(* CODESYS project TU München_Base.project

Project tree, tasks and I/O mapping:
  Device : CODESYS Control Win V3, 3S - Smart Software Solutions GmbH, order no. 305021, version 3.5.10.0
    application project
      libraries: Tc2_Standard, 3.3.1.0 (Beckhoff Automation GmbH); Tc2_System, 3.4.14.0 (Beckhoff Automation GmbH); Tc3_Interfaces, 3.4.2.0 (Beckhoff Automation GmbH); Tc3_Module, 3.3.11.0 (Beckhoff Automation GmbH)
      task PlcTask (cyclic, interval t#200ms, priority 22) calls MAIN
      GVLs/
        global variables GVL
      POUs/
        OMAC/
          Data Structures/
            Enum/
              data type TDataType
              data type TDiagnosisState
              data type TOperation
              data type TOperationState
              data type TPositionTable
            Condition/
              function block Condition [ST]: value, name
          OMAC_PackML_State_Machine/
            Enums/
              data type State
            Function Blocks/
              function block UnitMode [ST]: Reset, Stop, Hold, Enter, Suspend, AllowsEntering, ActingStateCompleted, UnSuspend, Clear, Start, UnHold, NextState, Abort, AllowsLeaving, Name, SupportedStates, CurrentState, Active
              function block UnitModeManager [ST]: Register, FindMode, SwitchUnitMode, AllowsSwitchingTo, ActiveUnitModeNumber, ActiveUnitMode
              function block Test [ST]
            Interfaces/
              interface IUnitMode: Stop, Hold, Unhold, Abort, NextState, Suspend, Start, ActingStateCompleted, AllowsEntering, UnSuspend, Enter, Reset, Clear, Name, CurrentState, Active, AllowsLeaving, SupportedStates
              interface IPlant
          Interface/
            interface IModule: resetting, completing, starting, holding, aborting, unHolding, stopping, clearing, execute
        program MAIN [ST]
        CM/
          function block Conveyor1 [ST]: transportWPToRamp1, holding, clearing, aborting, resetting, completing, stopping, starting, execute, transportWPToStart, unHolding
          function block Crane [ST]: turnLeftToStack, unHolding, lift, clearing, completing, execute, starting, turnRightToStack, turnRightToStamp, intake, turnLeftToConveyor, turnRightToConveyor, lower, turnLeftToStamp, holding, stopping, aborting, resetting, release
          function block Stack [ST]: offer, resetting, release, aborting, clearing, holding, completing, wait, starting, unHolding, stopping, execute
          function block Stamp [ST]: wait, clearing, lower, offer, lift, aborting, starting, resetting, execute, completing, unHolding, holding, stopping, release
        ConditionObserver/
          function block ConditionObserver [ST]: addPositivePrecondition, addNegativePreAndPostcondition, addPositivePostcondition, addCondition, checkConditions, addObjectsFromBuffer
        DiagnosisModul/
          function block DiagnosisModule [ST]: executeFailureDiagnois
        EM/
          function block SortingPlant [ST]: execute, unHolding, aborting, stopping, completing, clearing, starting, resetting, holding
          function block StampingPlant [ST]: holding, aborting, resetting, unHolding, clearing, completing, stopping, starting, execute
        UN/
          function block PickAndPlaceUnit [ST]: resetting, execute, completing, starting, holding, aborting, unHolding, clearing, stopping
*)

// Device/project/POUs/OMAC/Data Structures/Enum/TDataType
{attribute 'strict' := ''}
TYPE TDataType :
(
	tGRAPH := 0,
	tOPERATION := 1
);
END_TYPE

// Device/project/POUs/OMAC/Data Structures/Enum/TDiagnosisState
TYPE TDiagnosisState :
(
	tNODIAGNOSISSTATE := 0,
	tDIAGNOSISSTEP1,
	tDIAGNOSISSTEP2,
	tDIAGNOSISSTEP3,
	tDIAGNOSISSTEP4,
	tDIAGNOSISSTEP5,
	tDIAGNOSISFINISHED
);
END_TYPE

// Device/project/POUs/OMAC/Data Structures/Enum/TOperation
TYPE TOperation :
(
	tOPERATING := 0,
	tFINISHED := 1,
	tERROR := 2,
	tNORESPONSE := 3
);
END_TYPE

// Device/project/POUs/OMAC/Data Structures/Enum/TOperationState
TYPE TOperationState :
(
	tNOSTATE := 0,
	tSTACKEXTENDCYLINDER,
	tSTACKRETRACTCYLINDER,
	tSTACKWAITFOREXTEND,
	tCRANELOWERATSTACK,
	tCRANEINTAKE,
	tCRANELIFTATSTACK,
	tCRANETURNTOSTAMP,
	tCRANELOWERATSTAMP,
	tCRANERELEASE,
	tCRANELIFTATSTAMP,
	tCRANETURNTOCONVEYOR,
	tCRANELOWERATCONVEYOR,
	tCRANELIFTATCONVEYOR,
	tSTAMPRELEASE,
	tSTAMPLOWER,
	tSTAMPWAIT,
	tSTAMPLIFT,
	tSTAMPOFFER,
	tSTAMPINGPLANTTRANSPORTWPTOSTAMP,
	tSTAMPINGPLANTPROVIDEWP,
	tSTAMPINGPLANTSTAMPWP,
	tSTAMPINGPLANTTRANSPORTWPTOCONVEYOR,
	tCONVEYOR1TRANSPORTWPTORAMP1,
	tSORTINGPLANTTRANSPORTWPTORAMP,
	tPPUSTAMPWP,
	tPPUSORTWP,
	tOPERATIONFINISHED
);
END_TYPE

// Device/project/POUs/OMAC/Data Structures/Enum/TPositionTable
TYPE TPositionTable :
(
	NOPOSITION := 0,
	POSITION1,
	POSITION2,
	POSITION3,
	POSITION4,
	POSITION5,
	POSITION6,
	POSITION7,
	POSITION8
);
END_TYPE

// Device/project/POUs/OMAC/OMAC_PackML_State_Machine/Enums/State
/// Machine states
TYPE State :
(
	/// Bit 0
	Stopped := 16#1,
	/// Bit 1
	Resetting := 16#2,
	/// Bit 2
	Idle := 16#4,
	/// Bit 3
	Starting := 16#8,
	/// Bit 4
	Execute := 16#10,
	/// Bit 5
	Holding := 16#20,
	/// Bit 6
	Held := 16#40,
	/// Bit 7
	UnHolding := 16#80,
	/// Bit 8
	Suspending := 16#100,
	/// Bit 9
	Suspended := 16#200,
	/// Bit 10
	UnSuspending := 16#400,
	/// Bit 11
	Completing := 16#800,
	/// Bit 12
	Complete := 16#1000,
	/// Bit 13
	Stopping := 16#2000,
	/// Bit 14
	Aborting := 16#4000,
	/// Bit 15
	Aborted := 16#8000,
	/// Bit 16
	Clearing := 16#10000,
	No := 0,
	All := 16#1FFFF,
	Invalid := 16#80000000
) DWORD;
END_TYPE

// Device/project/GVLs/GVL
VAR_GLOBAL
	in_MagazinStartknopf : BOOL;
	in_MagazinNotaus : BOOL;
	in_MagazinSchieberAusgefahren : BOOL;
	in_MagazinSchieberNichtAusgefahren : BOOL;
	in_MagazinInduktiverSensor : BOOL;
	in_MagazinOptischerSensor : BOOL;
	in_MagazinWerkstueckGriffbereit : BOOL;
	
	in_KranAngesaugt : BOOL;
	in_KranUnten : BOOL;
	in_KranOben : BOOL;
	in_KranZeigtAufStempel : BOOL;
	in_KranZeigtAufLaufband : BOOL;
	in_KranZeigtAufMagazin : BOOL;
	
	in_StempelSchieberAusgefahren  : BOOL;
	in_StempelSchieberEingefahren  : BOOL;
	in_StempelWerkstueckVorhanden  : BOOL;
	in_StempelOben  : BOOL;
	in_StempelUnten  : BOOL;
	
	in_Sortierband_LichttasterKranInterface  : BOOL;
	in_Sortierband_KapazitiverSensorKranInterface  : BOOL;
	in_Sortierband_InduktiverSensorPusher1  : BOOL;
	in_Sortierband_LichttasterPusher1  : BOOL;
	in_Sortierband_InduktiverSensorPusher2  : BOOL;
	in_Sortierband_LichttasterPusher2  : BOOL;
	in_Sortierband_LichttasterSlide3  : BOOL;
	in_Sortierband_Pusher1Ausgefahren  : BOOL;
	in_Sortierband_Pusher1Eingefahren  : BOOL;
	in_Sortierband_Pusher2Ausgefahren  : BOOL;
	in_Sortierband_Pusher2Eingefahren  : BOOL;
	in_Sortierband_Lichtschranke3  : BOOL;
	
	in_Magazin_SchalterManAuto  : BOOL;
	
	out_MagazinSchieber : BOOL;
	
	out_KranSenken : BOOL;
	out_KranVakuumAn : BOOL;
	out_KranDreheRechts : BOOL;
	out_KranDreheLinks : BOOL;
	
	out_StempelSchieberAusfahren  : BOOL;
	out_StempelSchieberEinfahren  : BOOL;
	out_StempelStempeln  : BOOL;
	out_StempelStempelnDruck  : INT;
	
	out_SortierbandDreheVorwaerts  : BOOL;
	out_SortierbandDreheRueckwaerts  : BOOL;
	
	out_SortierbandPusher1  : BOOL;
	out_SortierbandPusher2  : BOOL;
	
	test_Sicherheitstuer_start : BOOL;
	test_Sicherheitstuer_auto_manuell : BOOL;
	
	test_test2  : BOOL;
	
	
	//virtual sensors
	v_MagazinWarten : BOOL;
	v_KranAngesaugt : BOOL;
	
	// ConditionObserver
	m_conditionObserver : ConditionObserver;
	m_condPropertyNames : ARRAY[1..30] OF STRING;
	m_condPropertyValues : ARRAY[1..30] OF BOOL;
	m_counterNewConditions : INT := 0;
	m_deleteConditions : BOOL;
	
	m_isReadingInformation : BOOL := FALSE;
	m_condPropertyNamesBuffer : ARRAY[1..30] OF STRING;
	m_condPropertyValuesBuffer : ARRAY[1..30] OF BOOL;
	m_counterNewConditionsBuffer : INT := 0;
	
	m_isFailure : BOOL;
	m_failurePart : STRING;
	m_failureRecoveryStrategy : STRING;
	m_isFailureMessage : BOOL;
	m_failureMessage : STRING;
	m_startDiagnosis : BOOL;
	m_startRecovery : BOOL;
	m_recoveryFinished : BOOL;
	m_restartProduction : BOOL;
	m_productionStarted : BOOL;
	
	m_startingFinished : BOOL;
	
	
	m_Conveyor1WPBeforePusher1 : BOOL;
	
	test_OMACState : STRING;

	
END_VAR

VAR_GLOBAL CONSTANT
	
	gc_usiMaxModes : USINT := 10;
	gc_maxObjectsArray : USINT := 10;
	
END_VAR

// Device/project/POUs/MAIN
/// Implementation of the OMAC State Machine
PROGRAM MAIN
VAR
	xInit : BOOL;
	
	productionUnitMode : UnitMode;
	currentUnitMode : IUnitMode;
	UnitModeManager : UnitModeManager;
		
	pickAndPlaceUnit : PickAndPlaceUnit;
	
	diagnosisModule : DiagnosisModule;
	
	m_StartButton : BOOL;
	lastStartButtonValue : BOOL;
	
	waitTON : TON;
	
END_VAR

IF NOT xInit THEN
	productionUnitMode(		sName:='Production_Mode',
							dwSupportedStates:=State.All,
							dwAllowsLeavingFromStates:=State.Execute,
							dwAllowsEnteringIntoStates:=State.Execute,
							eInitialState:=State.Idle,
							xActive:=TRUE);
	
	unitModeManager.Register(productionUnitMode);
	xInit := TRUE;
END_IF
currentUnitMode := unitModeManager.ActiveUnitMode;

// buttons
IF in_MagazinStartknopf AND NOT lastStartButtonValue THEN
	m_StartButton := TRUE;
ELSE
	m_StartButton := FALSE;
END_IF

//Condition Observer
m_conditionObserver.checkConditions(); //check if conditions are read

IF m_counterNewConditionsBuffer > 0 AND NOT m_isReadingInformation THEN
	m_conditionObserver.addObjectsFromBuffer();
END_IF


// OMAC STATE MACHINE
CASE currentUnitMode.CurrentState OF
	State.Idle:
		IF m_StartButton THEN
			currentUnitMode.Start();
		END_IF
	State.Starting:
		IF pickAndPlaceUnit.starting() = tFINISHED THEN
			currentUnitMode.ActingStateCompleted();
		END_IF
	State.Execute:
		IF m_isFailure THEN
			currentUnitMode.Hold();
		ELSIF pickAndPlaceUnit.execute() = tFINISHED THEN
			currentUnitMode.ActingStateCompleted();
		END_IF
	State.Holding:
		m_productionStarted := FALSE;
		IF pickAndPlaceUnit.holding() = tFINISHED THEN
			IF m_startDiagnosis THEN
				IF diagnosisModule.executeFailureDiagnois() = tFINISHED THEN
					currentUnitMode.ActingStateCompleted();
				END_IF
			END_IF
		END_IF
	State.Held:
		IF m_StartButton AND m_startRecovery THEN
			currentUnitMode.Unhold();
		END_IF
	State.UnHolding:
		IF pickAndPlaceUnit.unHolding(m_failureRecoveryStrategy) = tFINISHED THEN
			m_recoveryFinished := TRUE;
			IF m_restartProduction THEN
				m_isFailure := FALSE;
				m_failurePart := '';
				m_failureRecoveryStrategy := '';
				m_isFailureMessage := FALSE;
				m_failureMessage := '';
				m_startDiagnosis := FALSE;
				currentUnitMode.ActingStateCompleted();
			END_IF
		END_IF
	State.Completing:
		waitTON(IN:=TRUE,PT:=T#500MS);
		IF waitTON.Q THEN
			IF pickAndPlaceUnit.completing() = tFINISHED THEN
				currentUnitMode.ActingStateCompleted();
			END_IF
		END_IF	
	State.Complete:
		waitTON(IN:=FALSE,PT:=T#500MS);
		currentUnitMode.Reset();
	State.Resetting:
		test_OMACState := 'RESETTING';
		m_startRecovery := FALSE;
		m_recoveryFinished := FALSE;
		m_restartProduction := FALSE;
		m_productionStarted := FALSE;
		m_startingFinished := FALSE;
		IF pickAndPlaceUnit.resetting() = tFINISHED THEN
			currentUnitMode.ActingStateCompleted();
		END_IF
	State.Aborting:
	State.Aborted:	
	State.Clearing:
	State.Stopped:	
	State.Stopping:
END_CASE


lastStartButtonValue := in_MagazinStartknopf;

END_PROGRAM

// Device/project/POUs/OMAC/OMAC_PackML_State_Machine/Function Blocks/UnitModeManager
/// Function block to switch the current unit mode.
FUNCTION_BLOCK UnitModeManager
VAR
	apum: ARRAY[1..gc_usiMaxModes] OF IUnitMode;
	usiNumberOfUMs: USINT := 0;
	usiActualUM: USINT;
END_VAR

/// Registers an unit mode
METHOD Register : BOOL
VAR_INPUT
	pum: IUnitMode;
END_VAR
IF usiNumberOfUMs < gc_usiMaxModes THEN
	usiNumberOfUMs := usiNumberOfUMs + 1;
	apum[usiNumberOfUMs] := pum;
	IF usiActualUM = 0 THEN
		usiActualUM := 1;
		apum[usiNumberOfUMs].Active := TRUE;
	ELSE
		apum[usiNumberOfUMs].Active := FALSE;
	END_IF
	Register := TRUE;
END_IF
END_METHOD

/// Finds an unit mode by name.
{attribute 'hide' := ''}
{attribute 'object_name' := 'FindMode'}
METHOD PRIVATE FindMode : USINT
VAR_INPUT
	/// Name od the unit mode
	sName: STRING;
END_VAR
VAR
	usi: USINT;
END_VAR
FOR usi := 1 TO usiNumberOfUMs DO
	IF sName = apum[usi].Name THEN
		FindMode := usi;
		RETURN;
	END_IF
END_FOR
FindMode := gc_usiMaxModes+1;
END_METHOD

/// Switch to an other unit mode and check the permission.
/// Returns true if switching is allowed, returns false if switching is forbidden.
METHOD SwitchUnitMode : BOOL
VAR_INPUT
	/// Name of the unit mode to switch
	sNewModeName: STRING;
END_VAR
VAR
	pnew: POINTER TO UnitMode;
	usi: USINT;
END_VAR
usi := FindMode(sNewModeName);
SwitchUnitMode := FALSE;
IF usi>gc_usiMaxModes THEN
	RETURN;
END_IF

IF usi=usiActualUM THEN
	SwitchUnitMode := TRUE;
	RETURN;
END_IF

IF apum[usiActualUM].AllowsLeaving AND apum[usi].AllowsEntering(ActiveUnitMode.CurrentState) THEN
	apum[usi].Enter(ActiveUnitMode.CurrentState);
	apum[usiActualUM].Active := FALSE;
	apum[usi].Active := TRUE;
	usiActualUM := usi;
	SwitchUnitMode := TRUE;
END_IF
END_METHOD

/// Checks if the current state allows switching the current unit mode.
{attribute 'hide' := ''}
{attribute 'object_name' := 'AllowsSwitchingTo'}
METHOD PRIVATE AllowsSwitchingTo : BOOL
VAR_INPUT
	/// Unit mode to switch
	usi: USINT;
END_VAR
IF usi=usiActualUM THEN
	AllowsSwitchingTo := TRUE;
ELSE
	AllowsSwitchingTo := apum[usiActualUM].AllowsLeaving AND apum[usi].AllowsEntering(ActiveUnitMode.CurrentState);
END_IF
END_METHOD

{attribute 'monitoring' := 'variable'}
PROPERTY ActiveUnitModeNumber : USINT
GET
ActiveUnitModeNumber := usiActualUM;
END_GET
END_PROPERTY

/// Get and set the active unit mode.
PROPERTY ActiveUnitMode : IUnitMode
GET
ActiveUnitMode := apum[usiActualUM];
END_GET
END_PROPERTY

END_FUNCTION_BLOCK

// Device/project/POUs/OMAC/OMAC_PackML_State_Machine/Interfaces/IUnitMode
INTERFACE IUnitMode

{attribute 'object_name' := 'Stop'}
METHOD Stop : BOOL
END_METHOD

{attribute 'object_name' := 'Hold'}
METHOD Hold : BOOL
END_METHOD

{attribute 'object_name' := 'Unhold'}
METHOD Unhold : BOOL
END_METHOD

{attribute 'object_name' := 'Abort'}
METHOD Abort : BOOL
END_METHOD

{attribute 'object_name' := 'NextState'}
METHOD NextState : State
VAR_INPUT
	e: State;
END_VAR
END_METHOD

{attribute 'object_name' := 'Suspend'}
METHOD Suspend : BOOL
END_METHOD

{attribute 'object_name' := 'Start'}
METHOD Start : BOOL
END_METHOD

{attribute 'object_name' := 'ActingStateCompleted'}
METHOD ActingStateCompleted : BOOL
END_METHOD

{attribute 'object_name' := 'AllowsEntering'}
METHOD AllowsEntering : BOOL
VAR_INPUT
	e: State;
END_VAR
END_METHOD

{attribute 'object_name' := 'UnSuspend'}
METHOD UnSuspend : BOOL
END_METHOD

{attribute 'object_name' := 'Enter'}
METHOD Enter : BOOL
VAR_INPUT
	e: State;
END_VAR
END_METHOD

{attribute 'object_name' := 'Reset'}
METHOD Reset : BOOL
END_METHOD

{attribute 'object_name' := 'Clear'}
METHOD Clear : BOOL
END_METHOD

PROPERTY Name : STRING
GET
END_GET
END_PROPERTY

PROPERTY CurrentState : State
GET
END_GET
END_PROPERTY

PROPERTY Active : BOOL
GET
END_GET
SET
END_SET
END_PROPERTY

PROPERTY AllowsLeaving : BOOL
GET
END_GET
END_PROPERTY

PROPERTY SupportedStates : DWORD
GET
END_GET
END_PROPERTY

END_INTERFACE

// Device/project/POUs/OMAC/OMAC_PackML_State_Machine/Function Blocks/UnitMode
/// This function block describes an unit mode with all possible machine states, actions and the current state. 
/// The transition between unit modes is handled by the UnitModeMangager. 
{attribute 'hide_all_locals' := ''}
FUNCTION_BLOCK UnitMode IMPLEMENTS IUnitMode
VAR_INPUT
	/// Name of the unit mode
	sName: STRING;
	/// Supported states
	dwSupportedStates: DWORD := 2#11111111111111111;
	/// Leaving state conditions
	dwAllowsLeavingFromStates: DWORD := (State.Stopped OR State.Aborted);
	/// Entering state conditions
	dwAllowsEnteringIntoStates: DWORD := (State.Stopped OR State.Aborted);
	/// Initialization state
	eInitialState: State;
	/// True if this unit mode is active
	xActive: BOOL;
END_VAR
VAR
	{attribute 'hide' := ''}
	eState: State := State.Invalid;
	{attribute 'hide' := ''}
	bInit: BOOL;
END_VAR

IF NOT bInit THEN
	bInit:=TRUE;
	eState := eInitialState;
END_IF

{attribute 'object_name' := 'Reset'}
METHOD Reset : BOOL
CASE eState OF
State.Complete,
State.Stopped:
	IF (State.Resetting AND SupportedStates) = 0 THEN
		Reset := FALSE;
		RETURN;
	END_IF
	eState := State.Resetting;
	Reset := TRUE;
END_CASE
END_METHOD

{attribute 'object_name' := 'Stop'}
METHOD Stop : BOOL
CASE eState OF
State.Resetting,
State.Idle,
State.Starting,
State.Execute,
State.Holding,
State.Held,
State.UnHolding,
State.Suspending,
State.Suspended,
State.UnSuspending,
State.Completing,
State.Complete:
	IF (State.Stopping AND SupportedStates) = 0 THEN
		Stop := FALSE;
		RETURN;
	END_IF
	eState := State.Stopping;
	Stop := TRUE;
END_CASE
END_METHOD

{attribute 'object_name' := 'Hold'}
METHOD Hold : BOOL
CASE eState OF
State.Execute:
	IF (State.Holding AND SupportedStates) = 0 THEN
		Hold := FALSE;
		RETURN;
	END_IF
	eState := State.Holding;
	Hold := TRUE;
END_CASE
END_METHOD

/// Enters the state.
{attribute 'object_name' := 'Enter'}
METHOD Enter : BOOL
VAR_INPUT
	e: State;
END_VAR
eState := e;
END_METHOD

{attribute 'object_name' := 'Suspend'}
METHOD Suspend : BOOL
CASE eState OF
State.Execute:
	IF (State.Suspending AND SupportedStates) = 0 THEN
		Suspend := FALSE;
		RETURN;
	END_IF
	eState := State.Suspending;
	Suspend := TRUE;
END_CASE
END_METHOD

/// Checks if the state allows entering.
{attribute 'hide' := ''}
{attribute 'object_name' := 'AllowsEntering'}
METHOD AllowsEntering : BOOL
VAR_INPUT
	e: State;
END_VAR
IF (e AND dwAllowsEnteringIntoStates) > 0 THEN
	AllowsEntering := TRUE;
END_IF
END_METHOD

/// This method should be called by the program if an action has been finished.
{attribute 'object_name' := 'ActingStateCompleted'}
METHOD ActingStateCompleted : BOOL
CASE eState OF
State.Holding,
State.UnHolding,
State.Starting,
State.Completing,
State.Resetting,
State.UnSuspending,
State.Suspending,
State.Aborting,
State.Stopping,
State.Clearing:
	IF (NextState(eState) AND SupportedStates) = 0 THEN
		ActingStateCompleted := FALSE;
		RETURN;
	END_IF
	eState := NextState(eState);
	ActingStateCompleted := TRUE;
	
State.Execute:
	IF (State.Completing AND SupportedStates) = 0 THEN
		ActingStateCompleted := FALSE;
		RETURN;
	END_IF
	eState := State.Completing;
	ActingStateCompleted := TRUE;
END_CASE

IF eState = State.Invalid THEN
	ActingStateCompleted := FALSE;
END_IF
END_METHOD

{attribute 'object_name' := 'UnSuspend'}
METHOD UnSuspend : BOOL
CASE eState OF
State.Suspended:
	IF (State.UnSuspending AND SupportedStates) = 0 THEN
		UnSuspend := FALSE;
		RETURN;
	END_IF
	eState := State.UnSuspending;
	UnSuspend := TRUE;
END_CASE
END_METHOD

{attribute 'object_name' := 'Clear'}
METHOD Clear : BOOL
CASE eState OF
State.Aborted:
	IF (State.Clearing AND SupportedStates) = 0 THEN
		Clear := FALSE;
		RETURN;
	END_IF
	eState := State.Clearing;
	Clear := TRUE;
END_CASE
END_METHOD

{attribute 'object_name' := 'Start'}
METHOD Start : BOOL
CASE eState OF
State.Idle:
	IF (State.Starting AND SupportedStates) = 0 THEN
		Start := FALSE;
		RETURN;
	END_IF
	eState := State.Starting;
	Start := TRUE;
END_CASE
END_METHOD

{attribute 'object_name' := 'UnHold'}
METHOD UnHold : BOOL
CASE eState OF
State.Held:
	IF (State.UnHolding AND SupportedStates) = 0 THEN
		UnHold := FALSE;
		RETURN;
	END_IF
	eState := State.UnHolding;
	UnHold := TRUE;
END_CASE
END_METHOD

/// Get the next machine state without checking the supported states.
{attribute 'object_name' := 'NextState'}
METHOD NextState : State
VAR_INPUT
	e: State;
END_VAR
CASE e OF
State.Stopped:
	NextState := State.Resetting;
State.Resetting:
	NextState := State.Idle;
State.Idle:
	NextState := State.Starting;
State.Starting:
	NextState := State.Execute;
State.Execute:
	NextState := State.Invalid;
State.Holding:
	NextState := State.Held;
State.Held:
	NextState := State.UnHolding;
State.UnHolding:
	NextState := State.Execute;
State.Suspending:
	NextState := State.Suspended;
State.Suspended:
	NextState := State.UnSuspending;
State.UnSuspending:
	NextState := State.Execute;
State.Completing:
	NextState := State.Complete;
State.Complete:
	NextState := State.Resetting;
State.Stopping:
	NextState := State.Stopped;
State.Aborting:
	NextState := State.Aborted;
State.Aborted:
	NextState := State.Clearing;
State.Clearing:
	NextState := State.Stopped;
END_CASE
END_METHOD

{attribute 'object_name' := 'Abort'}
METHOD Abort : BOOL
CASE eState OF
State.Stopped,
State.Resetting,
State.Idle,
State.Starting,
State.Execute,
State.Holding,
State.Held,
State.UnHolding,
State.Suspending,
State.Suspended,
State.UnSuspending,
State.Completing,
State.Complete,
State.Stopping,
State.Clearing:
	IF (State.Aborting AND SupportedStates) = 0 THEN
		Abort := FALSE;
		RETURN;
	END_IF
	eState := State.Aborting;
	Abort := TRUE;
END_CASE
END_METHOD

/// True if the current state of this unit mode allows to be leaved.
PROPERTY AllowsLeaving : BOOL
GET
IF (eState AND dwAllowsLeavingFromStates) > 0 THEN
	AllowsLeaving := TRUE;
END_IF
END_GET
END_PROPERTY

/// Get the name of the unit mode
PROPERTY Name : STRING
GET
Name := sName;
END_GET
END_PROPERTY

/// Get all supported states.
PROPERTY SupportedStates : DWORD
GET
SupportedStates := dwSupportedStates;
END_GET
END_PROPERTY

/// Get the current machine state
PROPERTY CurrentState : State
GET
CurrentState := eState;
END_GET
END_PROPERTY

/// True if this unit mode is active.
PROPERTY Active : BOOL
GET
Active := xActive;
END_GET
SET
xActive := Active;
END_SET
END_PROPERTY

END_FUNCTION_BLOCK

// Device/project/POUs/OMAC/Data Structures/Condition/Condition
FUNCTION_BLOCK Condition
VAR_INPUT
	in_Name: STRING;
	in_Value: BOOL;
END_VAR
VAR
	m_name: STRING;
	m_value: BOOL;
END_VAR

m_name := in_Name;
m_value := in_Value;

PROPERTY value : BOOL
GET
value := m_value;
END_GET
SET
m_value := value;
END_SET
END_PROPERTY

PROPERTY name : STRING
GET
name := m_name;
END_GET
SET
m_name := name;
END_SET
END_PROPERTY

END_FUNCTION_BLOCK

// Device/project/POUs/UN/PickAndPlaceUnit
FUNCTION_BLOCK PickAndPlaceUnit IMPLEMENTS IModule
VAR_INPUT
END_VAR
VAR_OUTPUT
END_VAR
VAR
	operationState : TOperationState;	

	operationStampWP : TOperation;
	operationSortWP : TOperation;

	stampingPlant : StampingPlant;
	sortingPlant : SortingPlant;
	
	
END_VAR

{attribute 'object_name' := 'resetting'}
METHOD resetting : TOperation
operationState  := tNOSTATE;
operationStampWP := tOPERATING;
operationSortWP := tOPERATING;

//IF m_counterNewConditions = 0 THEN
	IF (stampingPlant.resetting() = tFINISHED) AND (sortingPlant.resetting() = tFINISHED) THEN
		resetting := tFINISHED;
	ELSE
		resetting := tOPERATING;
	END_IF
//ELSE
//	resetting := tOPERATING;
//END_IF
END_METHOD

{attribute 'object_name' := 'execute'}
METHOD execute : TOperation
IF operationState = tNOSTATE THEN
	operationState := tPPUSTAMPWP;
	m_conditionObserver.addNegativePreAndPostcondition('PPUSortWP');
	m_conditionObserver.addPositivePrecondition('PPUStampWP');
ELSIF operationState = tPPUSTAMPWP AND operationStampWP = tFINISHED THEN
	operationState := tPPUSORTWP;
	m_conditionObserver.addPositivePostcondition('PPUStampWP');
	m_conditionObserver.addPositivePrecondition('PPUSortWP');
ELSIF operationState = tPPUSORTWP AND operationSortWP = tFINISHED THEN
	operationState := tOPERATIONFINISHED;
	m_conditionObserver.addNegativePreAndPostcondition('PPUStampWP');
	m_conditionObserver.addPositivePostcondition('PPUSortWP');
END_IF


IF operationState = tPPUSTAMPWP THEN
	operationStampWP := stampingPlant.execute();
ELSIF operationState = tPPUSORTWP THEN
	operationSortWP := sortingPlant.execute();
ELSIF operationState = tOPERATIONFINISHED THEN
	execute := tFINISHED;
END_IF
END_METHOD

{attribute 'object_name' := 'completing'}
METHOD completing : TOperation
completing := sortingPlant.completing();
END_METHOD

{attribute 'object_name' := 'starting'}
METHOD starting : TOperation
starting := stampingPlant.starting();
END_METHOD

{attribute 'object_name' := 'holding'}
METHOD holding : TOperation
IF stampingPlant.holding() = tFINISHED AND sortingPlant.holding() = tFINISHED THEN
	holding := tFINISHED;
ELSE
	holding := tOPERATING;
END_IF
END_METHOD

{attribute 'object_name' := 'aborting'}
METHOD aborting : TOperation
END_METHOD

{attribute 'object_name' := 'unHolding'}
METHOD unHolding : TOperation
VAR_INPUT
	in_recoveryStrategy	: STRING;
END_VAR
IF in_recoveryStrategy = 'Conveyor1TransportWPToRamp1_SensorNotWorking' OR in_recoveryStrategy = 'Conveyor1TransportWPToRamp1_FalseTimigPusher' THEN
	unHolding := sortingPlant.unHolding(in_recoveryStrategy);
END_IF
END_METHOD

{attribute 'object_name' := 'clearing'}
METHOD clearing : TOperation
END_METHOD

{attribute 'object_name' := 'stopping'}
METHOD stopping : TOperation
END_METHOD

END_FUNCTION_BLOCK

// Device/project/POUs/OMAC/Interface/IModule
INTERFACE IModule

{attribute 'object_name' := 'resetting'}
METHOD resetting : TOperation
END_METHOD

{attribute 'object_name' := 'completing'}
METHOD completing : TOperation
END_METHOD

{attribute 'object_name' := 'starting'}
METHOD starting : TOperation
END_METHOD

{attribute 'object_name' := 'holding'}
METHOD holding : TOperation
END_METHOD

{attribute 'object_name' := 'aborting'}
METHOD aborting : TOperation
END_METHOD

{attribute 'object_name' := 'unHolding'}
METHOD unHolding : TOperation
VAR_INPUT
	in_recoveryStrategy: STRING;
END_VAR
END_METHOD

{attribute 'object_name' := 'stopping'}
METHOD stopping : TOperation
END_METHOD

{attribute 'object_name' := 'clearing'}
METHOD clearing : TOperation
END_METHOD

{attribute 'object_name' := 'execute'}
METHOD execute : TOperation
END_METHOD

END_INTERFACE

// Device/project/POUs/EM/StampingPlant
FUNCTION_BLOCK StampingPlant IMPLEMENTS IModule
VAR_INPUT
END_VAR
VAR_OUTPUT
END_VAR
VAR


	stack : Stack;
	stamp : Stamp;
	crane : Crane;
	
	operationState : TOperationState;
	
	operationCrane1 : TOperation;
	operationCrane2 : TOperation;
	operationStack : TOperation;
	operationStamp : TOperation;
	
END_VAR

{attribute 'object_name' := 'holding'}
METHOD holding : TOperation
holding:= crane.holding();
END_METHOD

{attribute 'object_name' := 'aborting'}
METHOD aborting : TOperation
END_METHOD

{attribute 'object_name' := 'resetting'}
METHOD resetting : TOperation
operationState := tNOSTATE;
operationCrane1 := tOPERATING;
operationCrane2 := tOPERATING;
operationStack := tOPERATING;
operationStamp := tOPERATING;

IF (stack.resetting() = tFINISHED) AND (crane.resetting() = tFINISHED) AND (stamp.resetting() = tFINISHED) THEN
	resetting := tFINISHED;
ELSE
	resetting := tOPERATING;
END_IF
END_METHOD

{attribute 'object_name' := 'unHolding'}
METHOD unHolding : TOperation
VAR_INPUT
	in_recoveryStrategy	: STRING;
END_VAR
END_METHOD

{attribute 'object_name' := 'clearing'}
METHOD clearing : TOperation
END_METHOD

{attribute 'object_name' := 'completing'}
METHOD completing : TOperation
END_METHOD

{attribute 'object_name' := 'stopping'}
METHOD stopping : TOperation
END_METHOD

{attribute 'object_name' := 'starting'}
METHOD starting : TOperation
IF (crane.starting() = tFINISHED) AND (stack.starting() = tFINISHED) AND (stamp.starting() = tFINISHED) THEN
	starting := tFINISHED;
ELSE
	starting := tOPERATING;
END_IF
END_METHOD

{attribute 'object_name' := 'execute'}
METHOD execute : TOperation
IF (operationState = tNOSTATE) THEN
	operationState := tSTAMPINGPLANTTRANSPORTWPTOSTAMP;
	m_conditionObserver.addNegativePreAndPostcondition('StampingPlantTransportWPToConveyor');
	m_conditionObserver.addPositivePrecondition('StampingPlantTransportWPToStamp');
ELSIF (operationState = tSTAMPINGPLANTTRANSPORTWPTOSTAMP) AND (operationCrane1 = tFINISHED) THEN
	operationState := tSTAMPINGPLANTPROVIDEWP;
	m_conditionObserver.addPositivePostcondition('StampingPlantTransportWPToStamp');
	m_conditionObserver.addPositivePrecondition('StampingPlantProvideWP');
ELSIF (operationState = tSTAMPINGPLANTPROVIDEWP) AND (operationStack = tFINISHED) THEN
	operationState := tSTAMPINGPLANTSTAMPWP;
	m_conditionObserver.addNegativePreAndPostcondition('StampingPlantTransportWPToStamp');
	m_conditionObserver.addPositivePostcondition('StampingPlantProvideWP');
	m_conditionObserver.addPositivePrecondition('StampingPlantStampWP');
ELSIF (operationState = tSTAMPINGPLANTSTAMPWP) AND (operationStamp = tFINISHED) THEN 
	operationState := tSTAMPINGPLANTTRANSPORTWPTOCONVEYOR;
	m_conditionObserver.addNegativePreAndPostcondition('StampingPlantProvideWP');
	m_conditionObserver.addPositivePostcondition('StampingPlantStampWP');
	m_conditionObserver.addPositivePrecondition('StampingPlantTransportWPToConveyor');
ELSIF (operationState = tSTAMPINGPLANTTRANSPORTWPTOCONVEYOR) AND (operationCrane2 = tFINISHED) THEN
	operationState := tOPERATIONFINISHED;
	m_conditionObserver.addNegativePreAndPostcondition('StampingPlantStampWP');
	m_conditionObserver.addPositivePostcondition('StampingPlantTransportWPToConveyor');
END_IF


IF operationState = tSTAMPINGPLANTTRANSPORTWPTOSTAMP THEN
	operationCrane1 := crane.execute('TransportWPToStamp');
ELSIF operationState = tSTAMPINGPLANTPROVIDEWP THEN
	operationStack := stack.execute();
ELSIF operationState = tSTAMPINGPLANTSTAMPWP THEN
	operationStamp := stamp.execute();
ELSIF operationState = tSTAMPINGPLANTTRANSPORTWPTOCONVEYOR THEN
	operationCrane2 := crane.execute('TransportWPToConveyor');
ELSIF operationState = tOPERATIONFINISHED THEN
	execute := tFINISHED;
END_IF
END_METHOD

END_FUNCTION_BLOCK

// Device/project/POUs/CM/Stack
FUNCTION_BLOCK Stack IMPLEMENTS IModule
VAR_INPUT
END_VAR
VAR_OUTPUT
END_VAR
VAR
	operationState : TOperationState;
	
	operationRelease : TOperation;
	operationWait : TOperation;
	operationOffer : TOperation;
	
	waitTon : TON;
END_VAR

METHOD offer : TOperation
VAR_INPUT
END_VAR
IF NOT in_MagazinSchieberAusgefahren THEN
	waitTon(IN:=FALSE, PT:=T#1S);
	out_MagazinSchieber := TRUE;
	offer := tOPERATING;
ELSE
	offer := tFINISHED;
END_IF
END_METHOD

{attribute 'object_name' := 'resetting'}
METHOD resetting : TOperation
operationState := tNOSTATE;

operationRelease := tOPERATING;
operationWait := tOPERATING;
operationOffer := tOPERATING;

resetting := tFINISHED;
END_METHOD

METHOD release : TOperation
VAR_INPUT
END_VAR
IF NOT in_MagazinSchieberNichtAusgefahren THEN
	out_MagazinSchieber := FALSE;
	release := tOPERATING;
ELSE
	release := tFINISHED;
END_IF
END_METHOD

{attribute 'object_name' := 'aborting'}
METHOD aborting : TOperation
END_METHOD

{attribute 'object_name' := 'clearing'}
METHOD clearing : TOperation
END_METHOD

{attribute 'object_name' := 'holding'}
METHOD holding : TOperation
END_METHOD

{attribute 'object_name' := 'completing'}
METHOD completing : TOperation
END_METHOD

METHOD wait : TOperation
VAR_INPUT
END_VAR
waitTon(IN:=TRUE, PT:=T#1S);
IF waitTon.Q THEN
	v_MagazinWarten := FALSE;
	wait := tFINISHED;
ELSE
	v_MagazinWarten := TRUE;
	wait := tOPERATING;
END_IF
END_METHOD

{attribute 'object_name' := 'starting'}
METHOD starting : TOperation
starting := THIS^.offer();
END_METHOD

{attribute 'object_name' := 'unHolding'}
METHOD unHolding : TOperation
VAR_INPUT
	in_recoveryStrategy	: STRING;
END_VAR
END_METHOD

{attribute 'object_name' := 'stopping'}
METHOD stopping : TOperation
END_METHOD

METHOD execute : TOperation
IF (operationState = tNOSTATE)  THEN
	operationState := tSTACKRETRACTCYLINDER;
	m_conditionObserver.addNegativePreAndPostcondition('StackOffer');
	m_conditionObserver.addPositivePrecondition('StackRelease');
ELSIF (operationState = tSTACKRETRACTCYLINDER) AND operationRelease = tFINISHED THEN
	operationState := tSTACKWAITFOREXTEND;
	m_conditionObserver.addPositivePostcondition('StackRelease');
	m_conditionObserver.addPositivePrecondition('StackWait');
ELSIF (operationState = tSTACKWAITFOREXTEND) AND operationWait = tFINISHED THEN
	operationState := tSTACKEXTENDCYLINDER;
	m_conditionObserver.addNegativePreAndPostcondition('StackRelease');
	m_conditionObserver.addPositivePostcondition('StackWait');
	m_conditionObserver.addPositivePrecondition('StackOffer');
ELSIF (operationState = tSTACKEXTENDCYLINDER) AND operationOffer = tFINISHED THEN
	operationState := tOPERATIONFINISHED;
	m_conditionObserver.addNegativePreAndPostcondition('StackWait');
	m_conditionObserver.addPositivePostcondition('StackOffer');
END_IF

IF operationState = tSTACKRETRACTCYLINDER THEN
	operationRelease := THIS^.release();
ELSIF operationState = tSTACKEXTENDCYLINDER THEN
	operationOffer := THIS^.offer();
ELSIF operationState = tSTACKWAITFOREXTEND THEN
	operationWait := THIS^.wait();
ELSIF operationState = tOPERATIONFINISHED THEN
	execute := tFINISHED;
END_IF
END_METHOD

END_FUNCTION_BLOCK

// Device/project/POUs/CM/Stamp
FUNCTION_BLOCK Stamp IMPLEMENTS IModule
VAR_INPUT
END_VAR
VAR_OUTPUT
END_VAR
VAR
	operationState : TOperationState;
	
	operationRelease : TOperation;
	operationLower : TOperation;
	operationWait : TOperation;
	operationLift : TOperation;
	operationOffer : TOperation;
	
	waitTon : TON;
END_VAR

METHOD wait : TOperation
VAR_INPUT
END_VAR
waitTon(IN:=TRUE, PT:=T#500MS);

IF waitTon.Q THEN
	wait := tFINISHED;
ELSE
	wait := tOPERATING;
END_IF
END_METHOD

{attribute 'object_name' := 'clearing'}
METHOD clearing : TOperation
END_METHOD

METHOD lower : TOperation
VAR_INPUT
END_VAR
IF NOT in_StempelUnten THEN
	out_StempelStempelnDruck := 4000;
	out_StempelStempeln := TRUE;
	lower := tOPERATING;
ELSE
	lower := tFINISHED;
END_IF
END_METHOD

METHOD offer : TOperation
VAR_INPUT
END_VAR
waitTon(IN:=FALSE, PT:=T#500MS);

IF NOT in_StempelSchieberAusgefahren THEN
	out_StempelSchieberAusfahren := TRUE;
	out_StempelSchieberEinfahren := FALSE;
	offer := tOPERATING;
ELSE
	offer := tFINISHED;
END_IF
END_METHOD

METHOD lift : TOperation
VAR_INPUT
END_VAR
IF NOT in_StempelOben THEN
	out_StempelStempeln := FALSE;
	out_StempelStempelnDruck := 0;
	lift := tOPERATING;
ELSE
	lift := tFINISHED;
END_IF
END_METHOD

{attribute 'object_name' := 'aborting'}
METHOD aborting : TOperation
END_METHOD

{attribute 'object_name' := 'starting'}
METHOD starting : TOperation
starting := offer();
END_METHOD

{attribute 'object_name' := 'resetting'}
METHOD resetting : TOperation
operationState := tNOSTATE;
	
operationRelease := tOPERATING;
operationLower := tOPERATING;
operationWait := tOPERATING;
operationLift := tOPERATING;
operationOffer := tOPERATING;

resetting := tFINISHED;
END_METHOD

{attribute 'object_name' := 'execute'}
METHOD execute : TOperation
IF (operationState = tNOSTATE) THEN
	operationState := tSTAMPRELEASE;
	m_conditionObserver.addNegativePreAndPostcondition('StampOffer');
	m_conditionObserver.addPositivePrecondition('StampRelease');
ELSIF (operationState = tSTAMPRELEASE) AND operationRelease = tFINISHED THEN
	operationState := tSTAMPLOWER;
	m_conditionObserver.addPositivePostcondition('StampRelease');
	m_conditionObserver.addPositivePrecondition('StampLower');
ELSIF operationState = tSTAMPLOWER AND operationLower = tFINISHED THEN
	operationState := tSTAMPWAIT;
	m_conditionObserver.addNegativePreAndPostcondition('StampRelease');
	m_conditionObserver.addPositivePostcondition('StampLower');
	m_conditionObserver.addPositivePrecondition('StampWait');
ELSIF operationState = tSTAMPWAIT AND operationWait = tFINISHED THEN
	operationState := tSTAMPLIFT;
	m_conditionObserver.addNegativePreAndPostcondition('StampLower');
	m_conditionObserver.addPositivePostcondition('StampWait');
	m_conditionObserver.addPositivePrecondition('StampLift');
ELSIF operationState = tSTAMPLIFT AND operationLift = tFINISHED THEN
	operationState := tSTAMPOFFER;
	m_conditionObserver.addNegativePreAndPostcondition('StampWait');
	m_conditionObserver.addPositivePostcondition('StampLift');
	m_conditionObserver.addPositivePrecondition('StampOffer');
ELSIF operationState = tSTAMPOFFER AND operationOffer = tFINISHED THEN
	operationState := tOPERATIONFINISHED;
	m_conditionObserver.addNegativePreAndPostcondition('StampLift');
	m_conditionObserver.addPositivePostcondition('StampOffer');
END_IF

IF operationState = tSTAMPRELEASE THEN
	operationRelease := THIS^.release();
ELSIF operationState = tSTAMPLOWER THEN
	operationLower := THIS^.lower();
ELSIF operationState = tSTAMPWAIT THEN
	operationWait := THIS^.wait();
ELSIF operationState = tSTAMPLIFT THEN
	operationLift := THIS^.lift();
ELSIF operationState = tSTAMPOFFER THEN
	operationOffer := THIS^.offer();
ELSIF operationState = tOPERATIONFINISHED THEN
	execute := tFINISHED;
END_IF
END_METHOD

{attribute 'object_name' := 'completing'}
METHOD completing : TOperation
END_METHOD

{attribute 'object_name' := 'unHolding'}
METHOD unHolding : TOperation
VAR_INPUT
	in_recoveryStrategy	: STRING;
END_VAR
END_METHOD

{attribute 'object_name' := 'holding'}
METHOD holding : TOperation
END_METHOD

{attribute 'object_name' := 'stopping'}
METHOD stopping : TOperation
END_METHOD

METHOD release : TOperation
VAR_INPUT
END_VAR
IF NOT in_StempelSchieberEingefahren THEN 
	out_StempelSchieberAusfahren := FALSE;
	out_StempelSchieberEinfahren := TRUE;
	release := tOPERATING;
ELSE
	release := tFINISHED;
END_IF
END_METHOD

END_FUNCTION_BLOCK

// Device/project/POUs/CM/Crane
FUNCTION_BLOCK Crane
VAR_INPUT
END_VAR
VAR_OUTPUT
END_VAR
VAR
	operationState : TOperationState;	
	operationState2 : TOperationState;	

	underPressureTON : TON;
	
	operationLowerAtStack : TOperation;
	operationIntake : TOperation;
	operationLiftAtStack : TOperation;
	operationTurnToStamp : TOperation;
	operationLowerAtStamp : TOperation;
	operationRelease : TOperation;
	operationLiftAtStamp : TOperation;
	
	operationTurnToConveyor : TOperation;
	operationLowerAtConveyor : TOperation;
	operationLiftAtConveyor : TOperation;
	
END_VAR

METHOD turnLeftToStack : TOperation
VAR_INPUT
END_VAR
IF NOT in_KranZeigtAufMagazin THEN
	out_KranDreheLinks := TRUE;
	turnLeftToStack := tOPERATING;
ELSE
	out_KranDreheLinks := FALSE;
	turnLeftToStack := tFINISHED;
END_IF
END_METHOD

{attribute 'object_name' := 'unHolding'}
METHOD unHolding : TOperation
VAR_INPUT
	in_recoveryStrategy	: STRING;
END_VAR
END_METHOD

METHOD lift : TOperation
VAR_INPUT
END_VAR
underPressureTON(IN:=FALSE, PT:=T#500MS);
IF NOT in_KranOben THEN
	out_KranSenken := FALSE;
	lift := tOPERATING;
ELSE
	lift := tFINISHED;
END_IF
END_METHOD

{attribute 'object_name' := 'clearing'}
METHOD clearing : TOperation
END_METHOD

{attribute 'object_name' := 'completing'}
METHOD completing : TOperation
END_METHOD

{attribute 'object_name' := 'execute'}
METHOD execute : TOperation
VAR_INPUT
	operationStrategy : STRING;
END_VAR
IF operationStrategy = 'TransportWPToStamp' THEN
	
	IF (operationState = tNOSTATE) AND in_KranOben AND in_KranZeigtAufMagazin AND NOT v_KranAngesaugt THEN
		operationState := tCRANELOWERATSTACK;
		m_conditionObserver.addNegativePreAndPostcondition('Crane1LiftAtStamp');
		m_conditionObserver.addPositivePrecondition('Crane1LowerAtStack');
	ELSIF (operationState = tCRANELOWERATSTACK) AND operationLowerAtStack = tFINISHED THEN
		operationState := tCRANEINTAKE;
		operationLowerAtStack := tOPERATING;
		m_conditionObserver.addPositivePostcondition('Crane1LowerAtStack');
		m_conditionObserver.addPositivePrecondition('Crane1Intake');
	ELSIF (operationState = tCRANEINTAKE) AND operationIntake = tFINISHED THEN
		operationState := tCRANELIFTATSTACK;
		operationIntake := tOPERATING;
		m_conditionObserver.addNegativePreAndPostcondition('Crane1LowerAtStack');
		m_conditionObserver.addPositivePostcondition('Crane1Intake');
		m_conditionObserver.addPositivePrecondition('Crane1LiftAtStack');
	ELSIF (operationState = tCRANELIFTATSTACK) AND operationLiftAtStack = tFINISHED THEN
		operationState := tCRANETURNTOSTAMP;
		operationLiftAtStack := tOPERATING;
		m_conditionObserver.addNegativePreAndPostcondition('Crane1Intake');
		m_conditionObserver.addPositivePostcondition('Crane1LiftAtStack');
		m_conditionObserver.addPositivePrecondition('Crane1TurnToStamp');
	ELSIF (operationState = tCRANETURNTOSTAMP) AND operationTurnToStamp = tFINISHED THEN
		operationState := tCRANELOWERATSTAMP;
		operationTurnToStamp := tOPERATING;
		m_conditionObserver.addNegativePreAndPostcondition('Crane1LiftAtStack');
		m_conditionObserver.addPositivePostcondition('Crane1TurnToStamp');
		m_conditionObserver.addPositivePrecondition('Crane1LowerAtStamp');
	ELSIF (operationState = tCRANELOWERATSTAMP) AND operationLowerAtStamp = tFINISHED THEN
		operationState := tCRANERELEASE;
		operationLowerAtStamp := tOPERATING;
		m_conditionObserver.addNegativePreAndPostcondition('Crane1TurnToStamp');
		m_conditionObserver.addPositivePostcondition('Crane1LowerAtStamp');
		m_conditionObserver.addPositivePrecondition('Crane1Release');
	ELSIF (operationState = tCRANERELEASE) AND operationRelease = tFINISHED THEN
		operationState := tCRANELIFTATSTAMP;
		operationRelease := tOPERATING;
		m_conditionObserver.addNegativePreAndPostcondition('Crane1LowerAtStamp');
		m_conditionObserver.addPositivePostcondition('Crane1Release');
		m_conditionObserver.addPositivePrecondition('Crane1LiftAtStamp');
	ELSIF (operationState = tCRANELIFTATSTAMP) AND operationLiftAtStamp = tFINISHED THEN
		operationState := tOPERATIONFINISHED;
		operationLiftAtStamp := tOPERATING;
		m_conditionObserver.addNegativePreAndPostcondition('Crane1Release');
		m_conditionObserver.addPositivePostcondition('Crane1LiftAtStamp');
	END_IF
	
	IF operationState = tCRANELOWERATSTACK THEN
		operationLowerAtStack := THIS^.lower();
	ELSIF operationState = tCRANELOWERATSTAMP THEN
		operationLowerAtStamp := THIS^.lower();
	ELSIF operationState = tCRANEINTAKE THEN
		operationIntake := THIS^.intake();
	ELSIF operationState = tCRANELIFTATSTACK THEN
		operationLiftAtStack := THIS^.lift();
	ELSIF operationState = tCRANELIFTATSTAMP THEN
		operationLiftAtStamp := THIS^.lift();
	ELSIF operationState = tCRANETURNTOSTAMP THEN
		operationTurnToStamp := THIS^.turnLeftToStamp();
	ELSIF operationState = tCRANERELEASE THEN
		operationRelease := THIS^.release();
	ELSIF operationState = tOPERATIONFINISHED THEN
		execute := tFINISHED;
	END_IF
	

ELSIF operationStrategy = 'TransportWPToConveyor' THEN
	
	IF (operationState2 = tNOSTATE) AND in_KranOben AND in_KranZeigtAufStempel AND NOT v_KranAngesaugt THEN
		operationState2 := tCRANELOWERATSTAMP;
		m_conditionObserver.addNegativePreAndPostcondition('Crane2LiftAtConveyor');
		m_conditionObserver.addPositivePrecondition('Crane2LowerAtStamp');
	ELSIF (operationState2 = tCRANELOWERATSTAMP) AND operationLowerAtStamp = tFINISHED THEN
		operationState2 := tCRANEINTAKE;
		operationLowerAtStamp := tOPERATING;
		m_conditionObserver.addPositivePostcondition('Crane2LowerAtStamp');
		m_conditionObserver.addPositivePrecondition('Crane2Intake');
	ELSIF (operationState2 = tCRANEINTAKE) AND operationIntake = tFINISHED THEN
		operationState2 := tCRANELIFTATSTAMP;
		operationIntake := tOPERATING;
		m_conditionObserver.addNegativePreAndPostcondition('Crane2LowerAtStamp');
		m_conditionObserver.addPositivePostcondition('Crane2Intake');
		m_conditionObserver.addPositivePrecondition('Crane2LiftAtStamp');
	ELSIF (operationState2 = tCRANELIFTATSTAMP) AND operationLiftAtStamp = tFINISHED THEN
		operationState2 := tCRANETURNTOCONVEYOR;
		operationLiftAtStamp := tOPERATING;
		m_conditionObserver.addNegativePreAndPostcondition('Crane2Intake');
		m_conditionObserver.addPositivePostcondition('Crane2LiftAtStamp');
		m_conditionObserver.addPositivePrecondition('Crane2TurnToConveyor');
	ELSIF (operationState2 = tCRANETURNTOCONVEYOR) AND operationTurnToConveyor = tFINISHED THEN
		operationState2 := tCRANELOWERATCONVEYOR;
		operationTurnToConveyor := tOPERATING;
		m_conditionObserver.addNegativePreAndPostcondition('Crane2LiftAtStamp');
		m_conditionObserver.addPositivePostcondition('Crane2TurnToConveyor');
		m_conditionObserver.addPositivePrecondition('Crane2LowerAtConveyor');
	ELSIF (operationState2 = tCRANELOWERATCONVEYOR) AND operationLowerAtConveyor = tFINISHED THEN
		operationState2 := tCRANERELEASE;
		operationLowerAtConveyor := tOPERATING;
		m_conditionObserver.addNegativePreAndPostcondition('Crane2TurnToConveyor');
		m_conditionObserver.addPositivePostcondition('Crane2LowerAtConveyor');
		m_conditionObserver.addPositivePrecondition('Crane2Release');
	ELSIF (operationState2 = tCRANERELEASE) AND operationRelease = tFINISHED THEN
		operationState2 := tCRANELIFTATCONVEYOR;
		operationRelease := tOPERATING;
		m_conditionObserver.addNegativePreAndPostcondition('Crane2LowerAtConveyor');
		m_conditionObserver.addPositivePostcondition('Crane2Release');
		m_conditionObserver.addPositivePrecondition('Crane2LiftAtConveyor');
	ELSIF (operationState2 = tCRANELIFTATCONVEYOR) AND operationLiftAtConveyor = tFINISHED THEN
		operationState2 := tOPERATIONFINISHED;
		operationLiftAtConveyor := tOPERATING;
		m_conditionObserver.addNegativePreAndPostcondition('Crane2Release');
		m_conditionObserver.addPositivePostcondition('Crane2LiftAtConveyor');
	END_IF
	
	IF operationState2 = tCRANELOWERATCONVEYOR THEN
		operationLowerAtConveyor := THIS^.lower();
	ELSIF operationState2 = tCRANELOWERATSTAMP THEN
		operationLowerAtStamp := THIS^.lower();
	ELSIF operationState2 = tCRANEINTAKE THEN
		operationIntake := THIS^.intake();
	ELSIF operationState2 = tCRANELIFTATCONVEYOR THEN
		operationLiftAtConveyor := THIS^.lift();
	ELSIF operationState2 = tCRANELIFTATSTAMP THEN
		operationLiftAtStamp := THIS^.lift();
	ELSIF operationState2 = tCRANETURNTOCONVEYOR THEN
		operationTurnToConveyor := THIS^.turnRightToConveyor();
	ELSIF operationState2 = tCRANERELEASE THEN
		operationRelease := THIS^.release();
	ELSIF operationState2 = tOPERATIONFINISHED THEN
		execute := tFINISHED;
	END_IF
	
	
	
END_IF
END_METHOD

{attribute 'object_name' := 'starting'}
METHOD starting : TOperation
starting := turnRightToStack();
END_METHOD

METHOD turnRightToStack : TOperation
VAR_INPUT
END_VAR
IF NOT in_KranZeigtAufMagazin THEN
	out_KranDreheRechts := TRUE;
	turnRightToStack := tOPERATING;
ELSE
	out_KranDreheRechts := FALSE;
	turnRightToStack := tFINISHED;
END_IF
END_METHOD

METHOD turnRightToStamp : TOperation
VAR_INPUT
END_VAR
IF NOT in_KranZeigtAufStempel THEN
	out_KranDreheRechts := TRUE;
	turnRightToStamp := tOPERATING;
ELSE
	out_KranDreheRechts := FALSE;
	turnRightToStamp := tFINISHED;
END_IF
END_METHOD

METHOD intake : TOperation
VAR_INPUT
END_VAR
underPressureTON(IN:=TRUE, PT:=T#500MS);
IF NOT in_KranAngesaugt OR NOT underPressureTON.Q THEN
	out_KranVakuumAn := TRUE;
	intake := tOPERATING;
ELSE
	v_KranAngesaugt := TRUE;
	intake := tFINISHED;
END_IF
END_METHOD

METHOD turnLeftToConveyor : TOperation
VAR_INPUT
END_VAR
IF NOT in_KranZeigtAufLaufband THEN
	out_KranDreheLinks := TRUE;
	turnLeftToConveyor := tOPERATING;
ELSE
	out_KranDreheLinks := FALSE;
	turnLeftToConveyor := tFINISHED;
END_IF
END_METHOD

METHOD turnRightToConveyor : TOperation
VAR_INPUT
END_VAR
IF NOT in_KranZeigtAufLaufband THEN
	out_KranDreheRechts := TRUE;
	turnRightToConveyor := tOPERATING;
ELSE
	out_KranDreheRechts := FALSE;
	turnRightToConveyor := tFINISHED;
END_IF
END_METHOD

METHOD lower : TOperation
VAR_INPUT
END_VAR
underPressureTON(IN:=FALSE, PT:=T#500MS);
IF NOT in_KranUnten THEN
	out_KranSenken := TRUE;
	lower := tOPERATING;
ELSE
	lower := tFINISHED;
END_IF
END_METHOD

METHOD turnLeftToStamp : TOperation
VAR_INPUT
END_VAR
IF NOT in_KranZeigtAufStempel THEN
	out_KranDreheLinks := TRUE;
	turnLeftToStamp := tOPERATING;
ELSE
	out_KranDreheLinks := FALSE;
	turnLeftToStamp := tFINISHED;
END_IF
END_METHOD

{attribute 'object_name' := 'holding'}
METHOD holding : TOperation
out_KranDreheLinks := FALSE;
out_KranDreheRechts := FALSE;
holding := tFINISHED;
END_METHOD

{attribute 'object_name' := 'stopping'}
METHOD stopping : TOperation
END_METHOD

{attribute 'object_name' := 'aborting'}
METHOD aborting : TOperation
END_METHOD

{attribute 'object_name' := 'resetting'}
METHOD resetting : TOperation
operationState := tNOSTATE;
operationState2 := tNOSTATE;
operationLowerAtStack := tOPERATING;
operationIntake  := tOPERATING;
operationLiftAtStack := tOPERATING;
operationTurnToStamp := tOPERATING;
operationLowerAtStamp := tOPERATING;
operationRelease := tOPERATING;
operationLiftAtStamp := tOPERATING;
operationTurnToConveyor := tOPERATING;
operationLowerAtConveyor := tOPERATING;
operationLiftAtConveyor := tOPERATING;

resetting := tFINISHED;
END_METHOD

METHOD release : TOperation
VAR_INPUT
END_VAR
underPressureTON(IN:=TRUE, PT:=T#500MS);
IF in_KranAngesaugt OR NOT underPressureTON.Q THEN
	out_KranVakuumAn := FALSE;
	release := tOPERATING;
ELSE
	v_KranAngesaugt := FALSE;
	release := tFINISHED;
END_IF
END_METHOD

END_FUNCTION_BLOCK

// Device/project/POUs/EM/SortingPlant
FUNCTION_BLOCK SortingPlant IMPLEMENTS IModule
VAR_INPUT
END_VAR
VAR_OUTPUT
END_VAR
VAR
	operationState : TOperationState;

	operationTransportWP : TOperation;	
	
	conveyor1 : Conveyor1;
	
	currentUnitMode : IUnitMode;
END_VAR

{attribute 'object_name' := 'execute'}
METHOD execute : TOperation
IF operationState = tNOSTATE THEN
	operationState := tSORTINGPLANTTRANSPORTWPTORAMP;
	m_conditionObserver.addPositivePrecondition('SortingPlantTransportWPToRamp');
ELSIF operationState = tSORTINGPLANTTRANSPORTWPTORAMP AND operationTransportWP = tFINISHED THEN
	operationState := tOPERATIONFINISHED;
	m_conditionObserver.addPositivePostcondition('SortingPlantTransportWPToRamp');
END_IF

IF operationState = tSORTINGPLANTTRANSPORTWPTORAMP THEN
	operationTransportWP := conveyor1.execute();
ELSIF operationState = tOPERATIONFINISHED THEN
	execute := tFINISHED;
END_IF
END_METHOD

{attribute 'object_name' := 'unHolding'}
METHOD unHolding : TOperation
VAR_INPUT
	in_recoveryStrategy	: STRING;
END_VAR
IF in_recoveryStrategy = 'Conveyor1TransportWPToRamp1_SensorNotWorking' OR in_recoveryStrategy = 'Conveyor1TransportWPToRamp1_FalseTimigPusher' THEN
	unHolding := conveyor1.unHolding(in_recoveryStrategy);
END_IF
END_METHOD

{attribute 'object_name' := 'aborting'}
METHOD aborting : TOperation
END_METHOD

{attribute 'object_name' := 'stopping'}
METHOD stopping : TOperation
END_METHOD

{attribute 'object_name' := 'completing'}
METHOD completing : TOperation
m_conditionObserver.addNegativePreAndPostcondition('SortingPlantTransportWPToRamp');
completing := conveyor1.completing();
END_METHOD

{attribute 'object_name' := 'clearing'}
METHOD clearing : TOperation
END_METHOD

{attribute 'object_name' := 'starting'}
METHOD starting : TOperation
END_METHOD

{attribute 'object_name' := 'resetting'}
METHOD resetting : TOperation
operationState := tNOSTATE;
operationTransportWP := tOPERATING;

resetting := conveyor1.resetting();
END_METHOD

{attribute 'object_name' := 'holding'}
METHOD holding : TOperation
holding := conveyor1.holding();
END_METHOD

END_FUNCTION_BLOCK

// Device/project/POUs/CM/Conveyor1
FUNCTION_BLOCK Conveyor1 IMPLEMENTS IModule
VAR_INPUT
END_VAR
VAR_OUTPUT
END_VAR
VAR
	operationState : TOperationState;
	
	operationTransportWP : TOperation;
	
	TONTransportWPToRamp1 : TON;
	m_ConveyorWPAtRamp1 : BOOL;
	
END_VAR

METHOD transportWPToRamp1 : TOperation
VAR_INPUT
END_VAR
transportWPToRamp1 := tOPERATING;
IF in_Sortierband_LichttasterPusher1 THEN
	m_Conveyor1WPBeforePusher1 := TRUE;
END_IF

IF in_Sortierband_Lichtschranke3 THEN
	m_ConveyorWPAtRamp1 := TRUE;
END_IF

IF NOT m_ConveyorWPAtRamp1 THEN
	out_SortierbandDreheVorwaerts := TRUE;
	
	IF m_Conveyor1WPBeforePusher1 THEN
		IF in_Magazin_SchalterManAuto THEN
			TONTransportWPToRamp1(IN:=TRUE,PT:=T#130MS);
		ELSE
			TONTransportWPToRamp1(IN:=TRUE,PT:=T#330MS);
		END_IF

		IF TONTransportWPToRamp1.Q THEN
			IF in_Sortierband_Pusher1Eingefahren THEN
				out_SortierbandPusher1 := TRUE;
			END_IF
		END_IF
	END_IF
END_IF

IF in_Sortierband_Pusher1Ausgefahren AND m_ConveyorWPAtRamp1 THEN
	out_SortierbandDreheVorwaerts := FALSE;
	out_SortierbandPusher1 := FALSE;
	transportWPToRamp1 := tFINISHED;
END_IF
END_METHOD

{attribute 'object_name' := 'holding'}
METHOD holding : TOperation
out_SortierbandDreheVorwaerts := FALSE;
out_SortierbandDreheRueckwaerts := FALSE;
out_SortierbandPusher1 := FALSE;
holding := tFINISHED;
END_METHOD

{attribute 'object_name' := 'clearing'}
METHOD clearing : TOperation
END_METHOD

{attribute 'object_name' := 'aborting'}
METHOD aborting : TOperation
END_METHOD

{attribute 'object_name' := 'resetting'}
METHOD resetting : TOperation
operationState := tNOSTATE;
operationTransportWP := tOPERATING;
TONTransportWPToRamp1(IN:=FALSE, PT:=T#1S);
m_Conveyor1WPBeforePusher1 := FALSE;
m_ConveyorWPAtRamp1 := FALSE;

resetting := tFINISHED;
END_METHOD

{attribute 'object_name' := 'completing'}
METHOD completing : TOperation
m_conditionObserver.addNegativePreAndPostcondition('Conveyor1TransportWPToRamp1');
completing := tFINISHED;
END_METHOD

{attribute 'object_name' := 'stopping'}
METHOD stopping : TOperation
END_METHOD

{attribute 'object_name' := 'starting'}
METHOD starting : TOperation
END_METHOD

{attribute 'object_name' := 'execute'}
METHOD execute : TOperation
IF operationState = tNOSTATE THEN
	operationState := tCONVEYOR1TRANSPORTWPTORAMP1;
	m_conditionObserver.addPositivePrecondition('Conveyor1TransportWPToRamp1');
ELSIF operationState = tCONVEYOR1TRANSPORTWPTORAMP1 AND operationTransportWP = tFINISHED THEN
	operationState := tOPERATIONFINISHED;
	m_conditionObserver.addPositivePostcondition('Conveyor1TransportWPToRamp1');
END_IF


IF operationState = tCONVEYOR1TRANSPORTWPTORAMP1 THEN
	operationTransportWP := THIS^.transportWPToRamp1();
ELSIF operationState = tOPERATIONFINISHED THEN
	execute := tFINISHED;
END_IF
END_METHOD

METHOD transportWPToStart : TOperation
VAR_INPUT
END_VAR
IF NOT in_Sortierband_LichttasterKranInterface THEN
	TONTransportWPToRamp1(IN:=FALSE,PT:=T#130MS);
	m_Conveyor1WPBeforePusher1 := FALSE;
	out_SortierbandDreheRueckwaerts := TRUE;
	transportWPToStart := tOPERATING;
ELSE
	out_SortierbandDreheRueckwaerts := FALSE;
	transportWPToStart := tFINISHED;
END_IF
END_METHOD

{attribute 'object_name' := 'unHolding'}
METHOD unHolding : TOperation
VAR_INPUT
	in_recoveryStrategy	: STRING;
END_VAR
IF in_recoveryStrategy = 'Conveyor1TransportWPToRamp1_SensorNotWorking' OR in_recoveryStrategy = 'Conveyor1TransportWPToRamp1_FalseTimigPusher' THEN
	unHolding := THIS^.transportWPToStart();
END_IF
END_METHOD

END_FUNCTION_BLOCK

// Device/project/POUs/DiagnosisModul/DiagnosisModule
FUNCTION_BLOCK DiagnosisModule
VAR_INPUT
END_VAR
VAR_OUTPUT
END_VAR
VAR
END_VAR

METHOD executeFailureDiagnois : TOperation
VAR_INPUT
END_VAR
executeFailureDiagnois := tOPERATING;

IF m_failurePart = 'Conveyor1TransportWPToRamp1' THEN
	IF NOT m_Conveyor1WPBeforePusher1 THEN
		m_failureRecoveryStrategy := 'Conveyor1TransportWPToRamp1_SensorNotWorking';
		m_isFailureMessage := TRUE;
		m_failureMessage := 'Sensor before Pusher not working!';
		executeFailureDiagnois := tFINISHED;
	ELSE
		m_failureRecoveryStrategy := 'Conveyor1TransportWPToRamp1_FalseTimigPusher';
		m_isFailureMessage := TRUE;
		m_failureMessage := 'Clean Conveyor!';
		executeFailureDiagnois := tFINISHED;
	END_IF
END_IF
END_METHOD

END_FUNCTION_BLOCK

// Device/project/POUs/ConditionObserver/ConditionObserver
FUNCTION_BLOCK ConditionObserver
VAR
	counterObjects: USINT := 0;
	propertyNames: ARRAY[1..30] OF STRING;
	propertyValues: ARRAY[1..30] OF BOOL;
END_VAR

{attribute 'object_name' := 'addPositivePrecondition'}
METHOD addPositivePrecondition
VAR_INPUT
	in_Name: STRING;
END_VAR
THIS^.addCondition(CONCAT('pre_',in_Name),TRUE);
THIS^.addCondition(CONCAT('post_',in_Name),FALSE);
END_METHOD

{attribute 'object_name' := 'addNegativePreAndPostcondition'}
METHOD addNegativePreAndPostcondition
VAR_INPUT
	in_Name: STRING;
END_VAR
THIS^.addCondition(CONCAT('pre_',in_Name),FALSE);
THIS^.addCondition(CONCAT('post_',in_Name),FALSE);
END_METHOD

{attribute 'object_name' := 'addPositivePostcondition'}
METHOD addPositivePostcondition
VAR_INPUT
	in_Name: STRING;
END_VAR
THIS^.addCondition(CONCAT('pre_',in_Name),FALSE);
THIS^.addCondition(CONCAT('post_',in_Name),TRUE);
END_METHOD

{attribute 'object_name' := 'addCondition'}
METHOD addCondition
VAR_INPUT
	in_Name: STRING;
	in_Value: BOOL;
END_VAR
IF NOT m_isReadingInformation THEN
	IF counterObjects < 30 THEN
		counterObjects := counterObjects + 1;
		propertyNames[counterObjects] := in_Name;
		propertyValues[counterObjects] := in_Value;
		m_counterNewConditions := counterObjects;
		m_condPropertyNames := propertyNames;
		m_condPropertyValues := propertyValues;
	END_IF
ELSE
	IF m_counterNewConditionsBuffer < 30 THEN
		m_counterNewConditionsBuffer := m_counterNewConditionsBuffer + 1;
		m_condPropertyNamesBuffer[m_counterNewConditionsBuffer] := in_Name;
		m_condPropertyValuesBuffer[m_counterNewConditionsBuffer] := in_Value;
	END_IF
END_IF
END_METHOD

{attribute 'object_name' := 'checkConditions'}
METHOD checkConditions
VAR
	i: INT;
END_VAR
IF m_deleteConditions THEN
	FOR i:=1 TO 30 BY 1 DO
		propertyNames[i] := '';
		propertyValues[i] := FALSE;
	END_FOR
	counterObjects := 0;
	m_counterNewConditions := 0;
	m_condPropertyNames := propertyNames;
	m_condPropertyValues := propertyValues;
	m_deleteConditions := FALSE;
END_IF
END_METHOD

{attribute 'object_name' := 'addObjectsFromBuffer'}
METHOD addObjectsFromBuffer
VAR
	i: INT;
END_VAR
FOR i:=1 TO m_counterNewConditionsBuffer BY 1 DO
	m_conditionObserver.addCondition(m_condPropertyNamesBuffer[i],m_condPropertyValuesBuffer[i]);
END_FOR
m_counterNewConditionsBuffer := 0;
END_METHOD

END_FUNCTION_BLOCK

// Device/project/POUs/OMAC/OMAC_PackML_State_Machine/Function Blocks/Test
FUNCTION_BLOCK Test
VAR_INPUT
END_VAR
VAR_OUTPUT
END_VAR
VAR	
	UnitModeManager : UnitModeManager;
	currentUnitMode : IUnitMode;
END_VAR


currentUnitMode := unitModeManager.ActiveUnitMode;
IF(currentUnitMode.CurrentState = State.Stopped)
	THEN RETURN;
END_IF

END_FUNCTION_BLOCK

// Device/project/POUs/OMAC/OMAC_PackML_State_Machine/Interfaces/IPlant
INTERFACE IPlant

END_INTERFACE
